# EPICS autosave request: roperApp/Db/roper_settings.req
file "ADBase_settings.req", "P=$(P), R=$(R)
file "NDFile_settings.req", "P=$(P), R=$(R)
$(P)$(R)NumAcquisitions
$(P)$(R)RoperShutterMode
$(P)$(R)AutoDataType
$(P)$(R)Temperature
$(P)$(R)UseBgd
$(P)$(R)BgdFileName
$(P)$(R)Comment1
$(P)$(R)Comment2
$(P)$(R)Comment3
$(P)$(R)Comment4
$(P)$(R)Comment5
